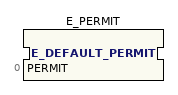
      [picture p24: application _02_Parameters.Ex4]
      FBS
        E_PERMIT : E_DEFAULT_PERMIT(PERMIT := 0);
      END_FBS
    END_SUBAPPLICATION
    SUBAPPLICATION Ex6 (* Any type: required casts  &#10; &#10;- Trigger REQ &#10;- Expect CNF and OUT:=13 *)
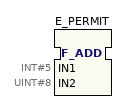
      FBS
        E_PERMIT : F_ADD(IN1 := INT#5, IN2 := UINT#8);
      END_FBS
    END_SUBAPPLICATION
    SUBAPPLICATION Ex5a (* integer parameter &#10; &#10;- Trigger REQ &#10;- Expect CNF, OUT:=5 *)
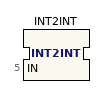
      FBS
        INT2INT : INT2INT(IN := 5);
      END_FBS
    END_SUBAPPLICATION
    SUBAPPLICATION Ex5b (* integer parameter with prefix &#10; &#10;- Trigger REQ &#10;- Expect CNF, OUT:=5 *)
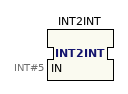
      FBS
        INT2INT : INT2INT(IN := INT#5);
      END_FBS
    END_SUBAPPLICATION
    SUBAPPLICATION Ex5c (* integer parameter with prefix (upcast) &#10; &#10;- Trigger REQ &#10;- Expect CNF, OUT:=5 *)
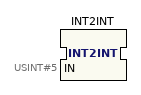
      FBS
        INT2INT : INT2INT(IN := USINT#5);
      END_FBS
    END_SUBAPPLICATION
  END_APPLICATION
  APPLICATION _04_DataWith
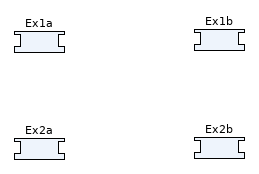
    (* Group Info_DataConnections: The subapps in this App serve as test cases for various versions of WITH-constructs (on updating data values to the outputs). &#10;- WITH at the inputs &#10;- WITH at the outputs *)
    SUBAPPLICATION Ex1a (* trigger REQ, expect CNF and &#10;DO1.OUT:=TRUE &#10;DO2.OUT:=-10 &#10;DO3.OUT:=15 &#10;DO4.OUT:=2.0 (data values from type) *)
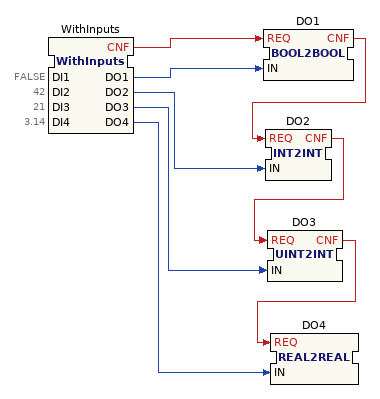
      FBS
        WithInputs : WithInputs(DI1 := FALSE, DI2 := 42, DI3 := 21, DI4 := 3.14);
        DO1 : BOOL2BOOL;
        DO2 : INT2INT;
        DO3 : UINT2INT;
        DO4 : REAL2REAL;
      END_FBS
      EVENT_CONNECTIONS
        WithInputs.CNF TO DO1.REQ;
        DO1.CNF TO DO2.REQ;
        DO2.CNF TO DO3.REQ;
        DO3.CNF TO DO4.REQ;
      END_CONNECTIONS
      DATA_CONNECTIONS
        WithInputs.DO1 TO DO1.IN;
        WithInputs.DO2 TO DO2.IN;
        WithInputs.DO3 TO DO3.IN;
        WithInputs.DO4 TO DO4.IN;
      END_CONNECTIONS
    END_SUBAPPLICATION
    SUBAPPLICATION Ex1b (* trigger UPDATE, expect CNF and &#10;DO1.OUT:=FALSE &#10;DO2.OUT:=42 &#10;DO3.OUT:=21 &#10;DO4.OUT:=3.14 (data values from type) *)
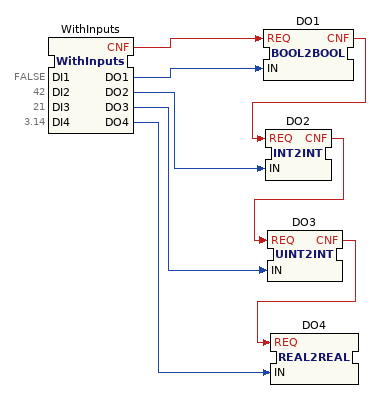
      FBS
        WithInputs : WithInputs(DI1 := FALSE, DI2 := 42, DI3 := 21, DI4 := 3.14);
        DO1 : BOOL2BOOL;
        DO2 : INT2INT;
        DO3 : UINT2INT;
        DO4 : REAL2REAL;
      END_FBS
      EVENT_CONNECTIONS
        WithInputs.CNF TO DO1.REQ;
        DO1.CNF TO DO2.REQ;
        DO2.CNF TO DO3.REQ;
        DO3.CNF TO DO4.REQ;
      END_CONNECTIONS
      DATA_CONNECTIONS
        WithInputs.DO1 TO DO1.IN;
        WithInputs.DO2 TO DO2.IN;
        WithInputs.DO3 TO DO3.IN;
        WithInputs.DO4 TO DO4.IN;
      END_CONNECTIONS
    END_SUBAPPLICATION
    SUBAPPLICATION Ex2a (* trigger REQ, expect CNF and &#10;DO1.OUT:=TRUE &#10;DO2.OUT:=-42 &#10;DO3.OUT:=21 &#10;DO4.OUT:=3.14 (data values from type) *)
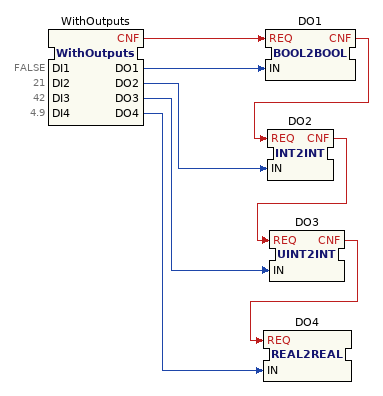
      FBS
        DO1 : BOOL2BOOL;
        DO2 : INT2INT;
        DO3 : UINT2INT;
        DO4 : REAL2REAL;
        WithOutputs : WithOutputs(DI1 := FALSE, DI2 := 21, DI3 := 42, DI4 := 4.9);
      END_FBS
      EVENT_CONNECTIONS
        DO1.CNF TO DO2.REQ;
        DO2.CNF TO DO3.REQ;
        DO3.CNF TO DO4.REQ;
        WithOutputs.CNF TO DO1.REQ;
      END_CONNECTIONS
      DATA_CONNECTIONS
        WithOutputs.DO1 TO DO1.IN;
        WithOutputs.DO2 TO DO2.IN;
        WithOutputs.DO3 TO DO3.IN;
        WithOutputs.DO4 TO DO4.IN;
      END_CONNECTIONS
    END_SUBAPPLICATION
    SUBAPPLICATION Ex2b (* trigger UPDATE, expect CNF and &#10;DO1.OUT:=FALSE &#10;DO2.OUT:=21 &#10;DO3.OUT:=42 &#10;DO4.OUT:=4.9 (data values from parameters) *)
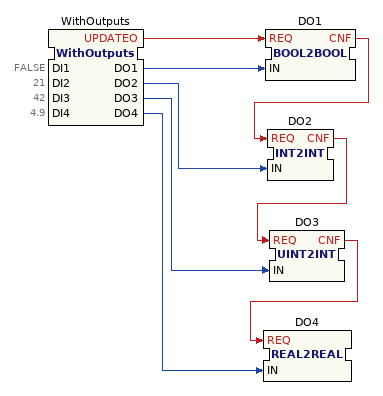
      FBS
        DO1 : BOOL2BOOL;
        DO2 : INT2INT;
        DO3 : UINT2INT;
        DO4 : REAL2REAL;
        WithOutputs : WithOutputs(DI1 := FALSE, DI2 := 21, DI3 := 42, DI4 := 4.9);
      END_FBS
      EVENT_CONNECTIONS
        DO1.CNF TO DO2.REQ;
        DO2.CNF TO DO3.REQ;
        DO3.CNF TO DO4.REQ;
        WithOutputs.UPDATEO TO DO1.REQ;
      END_CONNECTIONS
      DATA_CONNECTIONS
        WithOutputs.DO1 TO DO1.IN;
        WithOutputs.DO2 TO DO2.IN;
        WithOutputs.DO3 TO DO3.IN;
        WithOutputs.DO4 TO DO4.IN;
      END_CONNECTIONS
    END_SUBAPPLICATION
  END_APPLICATION
  APPLICATION _05_Adapter
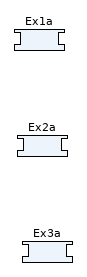
    (* Group Info_Adapter: The subapps in this App serve as test cases for various versions of WITH-constructs (on updating data values to the outputs). &#10;- WITH at the inputs &#10;- WITH at the outputs *)
    SUBAPPLICATION Ex1a (* Adapter with just events &#10;- trigger Fb1.REQ  &#10;- expect Fb1.CNF and Fb1.RSP *)
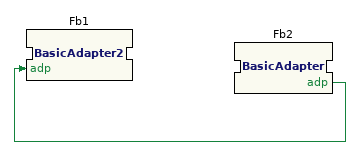
      FBS
        Fb1 : BasicAdapter2;
        Fb2 : BasicAdapter;
      END_FBS
      ADAPTER_CONNECTIONS
        Fb2.adp TO Fb1.adp;
      END_CONNECTIONS
    END_SUBAPPLICATION
    SUBAPPLICATION Ex2a (* Adapter with an event and data &#10;- trigger Fb1.REQ  &#10;- expect Fb2.CNF with Fb2.OUT:=TRUE *)
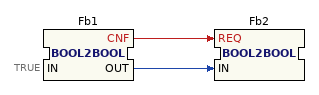
      FBS
        Fb1 : BOOL2BOOL(IN := TRUE);
        Fb2 : BOOL2BOOL;
      END_FBS
      EVENT_CONNECTIONS
        Fb1.CNF TO Fb2.REQ;
      END_CONNECTIONS
      DATA_CONNECTIONS
        Fb1.OUT TO Fb2.IN;
      END_CONNECTIONS
    END_SUBAPPLICATION
    SUBAPPLICATION Ex3a (* Adapter with a WITH (do not update all data) &#10;- trigger Fb1.REQ  &#10;- expect Fb2.CNF with Fb2.OUT:=TRUE *)
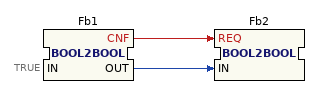
      FBS
        Fb1 : BOOL2BOOL(IN := TRUE);
        Fb2 : BOOL2BOOL;
      END_FBS
      EVENT_CONNECTIONS
        Fb1.CNF TO Fb2.REQ;
      END_CONNECTIONS
      DATA_CONNECTIONS
        Fb1.OUT TO Fb2.IN;
      END_CONNECTIONS
    END_SUBAPPLICATION
  END_APPLICATION
  DEVICE RaspberryPI : (MGR_ID := "localhost:61499")
    {SET_ATTRIBUTE(Profile, HOLOBLOC)}
    RESOURCE EMB_RES : 
    END_RESOURCE
  END_DEVICE
  SEGMENTS
    Ethernet_1 : ;
    Ethernet : ;
  END_SEGMENTS
END_SYSTEM
